afGe[0  , 0] := 1.00000E+01; afGe[0  , 1] := 8.81266E-03;
afGe[1  , 0] := 1.99800E+01; afGe[1  , 1] := 9.77619E-03;
afGe[2  , 0] := 2.99600E+01; afGe[2  , 1] := 9.38887E-01;
afGe[3  , 0] := 3.99400E+01; afGe[3  , 1] := 1.88885E+00;
afGe[4  , 0] := 4.99200E+01; afGe[4  , 1] := 3.37924E+00;
afGe[5  , 0] := 5.99000E+01; afGe[5  , 1] := 5.17287E+00;
afGe[6  , 0] := 6.98800E+01; afGe[6  , 1] := 6.99851E+00;
afGe[7  , 0] := 7.98600E+01; afGe[7  , 1] := 8.65575E+00;
afGe[8  , 0] := 8.98400E+01; afGe[8  , 1] := 1.00383E+01;
afGe[9  , 0] := 9.98200E+01; afGe[9  , 1] := 1.11123E+01;
afGe[10 , 0] := 1.09800E+02; afGe[10 , 1] := 1.18992E+01;
afGe[11 , 0] := 1.19780E+02; afGe[11 , 1] := 1.25300E+01;
afGe[12 , 0] := 1.29760E+02; afGe[12 , 1] := 1.31929E+01;
afGe[13 , 0] := 1.39740E+02; afGe[13 , 1] := 1.34683E+01;
afGe[14 , 0] := 1.49720E+02; afGe[14 , 1] := 1.35531E+01;
afGe[15 , 0] := 1.59700E+02; afGe[15 , 1] := 1.35254E+01;
afGe[16 , 0] := 1.69680E+02; afGe[16 , 1] := 1.34259E+01;
afGe[17 , 0] := 1.79660E+02; afGe[17 , 1] := 1.34620E+01;
afGe[18 , 0] := 1.89640E+02; afGe[18 , 1] := 1.35247E+01;
afGe[19 , 0] := 1.99620E+02; afGe[19 , 1] := 1.33231E+01;
afGe[20 , 0] := 2.09600E+02; afGe[20 , 1] := 1.30862E+01;
afGe[21 , 0] := 2.19580E+02; afGe[21 , 1] := 1.28308E+01;
afGe[22 , 0] := 2.29560E+02; afGe[22 , 1] := 1.25655E+01;
afGe[23 , 0] := 2.39540E+02; afGe[23 , 1] := 1.22951E+01;
afGe[24 , 0] := 2.49520E+02; afGe[24 , 1] := 1.20227E+01;
afGe[25 , 0] := 2.59500E+02; afGe[25 , 1] := 1.17524E+01;
afGe[26 , 0] := 2.69480E+02; afGe[26 , 1] := 1.14845E+01;
afGe[27 , 0] := 2.79460E+02; afGe[27 , 1] := 1.12208E+01;
afGe[28 , 0] := 2.89440E+02; afGe[28 , 1] := 1.09627E+01;
afGe[29 , 0] := 2.99420E+02; afGe[29 , 1] := 1.07107E+01;
afGe[30 , 0] := 3.09400E+02; afGe[30 , 1] := 1.04654E+01;
afGe[31 , 0] := 3.19380E+02; afGe[31 , 1] := 1.02271E+01;
afGe[32 , 0] := 3.29360E+02; afGe[32 , 1] := 9.99516E+00;
afGe[33 , 0] := 3.39340E+02; afGe[33 , 1] := 9.77038E+00;
afGe[34 , 0] := 3.49320E+02; afGe[34 , 1] := 9.55249E+00;
afGe[35 , 0] := 3.59300E+02; afGe[35 , 1] := 9.34153E+00;
afGe[36 , 0] := 3.69280E+02; afGe[36 , 1] := 9.13877E+00;
afGe[37 , 0] := 3.79260E+02; afGe[37 , 1] := 8.94103E+00;
afGe[38 , 0] := 3.89240E+02; afGe[38 , 1] := 8.75052E+00;
afGe[39 , 0] := 3.99220E+02; afGe[39 , 1] := 8.56542E+00;
afGe[40 , 0] := 4.09200E+02; afGe[40 , 1] := 8.38625E+00;
afGe[41 , 0] := 4.19180E+02; afGe[41 , 1] := 8.21293E+00;
afGe[42 , 0] := 4.29160E+02; afGe[42 , 1] := 8.04518E+00;
afGe[43 , 0] := 4.39140E+02; afGe[43 , 1] := 7.88279E+00;
afGe[44 , 0] := 4.49120E+02; afGe[44 , 1] := 7.72562E+00;
afGe[45 , 0] := 4.59100E+02; afGe[45 , 1] := 7.57349E+00;
afGe[46 , 0] := 4.69080E+02; afGe[46 , 1] := 7.42603E+00;
afGe[47 , 0] := 4.79060E+02; afGe[47 , 1] := 7.28323E+00;
afGe[48 , 0] := 4.89040E+02; afGe[48 , 1] := 7.14478E+00;
afGe[49 , 0] := 4.99020E+02; afGe[49 , 1] := 7.01042E+00;
afGe[50 , 0] := 5.09000E+02; afGe[50 , 1] := 6.87999E+00;
afGe[51 , 0] := 5.18980E+02; afGe[51 , 1] := 6.75328E+00;
afGe[52 , 0] := 5.28960E+02; afGe[52 , 1] := 6.63015E+00;
afGe[53 , 0] := 5.38940E+02; afGe[53 , 1] := 6.50950E+00;
afGe[54 , 0] := 5.48920E+02; afGe[54 , 1] := 6.37387E+00;
afGe[55 , 0] := 5.58900E+02; afGe[55 , 1] := 6.24150E+00;
afGe[56 , 0] := 5.68880E+02; afGe[56 , 1] := 6.11335E+00;
afGe[57 , 0] := 5.78860E+02; afGe[57 , 1] := 5.98927E+00;
afGe[58 , 0] := 5.88840E+02; afGe[58 , 1] := 5.86901E+00;
afGe[59 , 0] := 5.98820E+02; afGe[59 , 1] := 5.75252E+00;
afGe[60 , 0] := 6.08800E+02; afGe[60 , 1] := 5.63965E+00;
afGe[61 , 0] := 6.18780E+02; afGe[61 , 1] := 5.53035E+00;
afGe[62 , 0] := 6.28760E+02; afGe[62 , 1] := 5.42432E+00;
afGe[63 , 0] := 6.38740E+02; afGe[63 , 1] := 5.32161E+00;
afGe[64 , 0] := 6.48720E+02; afGe[64 , 1] := 5.22199E+00;
afGe[65 , 0] := 6.58700E+02; afGe[65 , 1] := 5.12538E+00;
afGe[66 , 0] := 6.68680E+02; afGe[66 , 1] := 5.03171E+00;
afGe[67 , 0] := 6.78660E+02; afGe[67 , 1] := 4.94078E+00;
afGe[68 , 0] := 6.88640E+02; afGe[68 , 1] := 4.85261E+00;
afGe[69 , 0] := 6.98620E+02; afGe[69 , 1] := 4.76709E+00;
afGe[70 , 0] := 7.08600E+02; afGe[70 , 1] := 4.68403E+00;
afGe[71 , 0] := 7.18580E+02; afGe[71 , 1] := 4.60334E+00;
afGe[72 , 0] := 7.28560E+02; afGe[72 , 1] := 4.52505E+00;
afGe[73 , 0] := 7.38540E+02; afGe[73 , 1] := 4.44896E+00;
afGe[74 , 0] := 7.48520E+02; afGe[74 , 1] := 4.37500E+00;
afGe[75 , 0] := 7.58500E+02; afGe[75 , 1] := 4.30316E+00;
afGe[76 , 0] := 7.68480E+02; afGe[76 , 1] := 4.23330E+00;
afGe[77 , 0] := 7.78460E+02; afGe[77 , 1] := 4.16541E+00;
afGe[78 , 0] := 7.88440E+02; afGe[78 , 1] := 4.09937E+00;
afGe[79 , 0] := 7.98420E+02; afGe[79 , 1] := 4.03513E+00;
afGe[80 , 0] := 8.08400E+02; afGe[80 , 1] := 3.97263E+00;
afGe[81 , 0] := 8.18380E+02; afGe[81 , 1] := 3.91191E+00;
afGe[82 , 0] := 8.28360E+02; afGe[82 , 1] := 3.85273E+00;
afGe[83 , 0] := 8.38340E+02; afGe[83 , 1] := 3.79513E+00;
afGe[84 , 0] := 8.48320E+02; afGe[84 , 1] := 3.73906E+00;
afGe[85 , 0] := 8.58300E+02; afGe[85 , 1] := 3.68448E+00;
afGe[86 , 0] := 8.68280E+02; afGe[86 , 1] := 3.63135E+00;
afGe[87 , 0] := 8.78260E+02; afGe[87 , 1] := 3.57961E+00;
afGe[88 , 0] := 8.88240E+02; afGe[88 , 1] := 3.52916E+00;
afGe[89 , 0] := 8.98220E+02; afGe[89 , 1] := 3.48008E+00;
afGe[90 , 0] := 9.08200E+02; afGe[90 , 1] := 3.43216E+00;
afGe[91 , 0] := 9.18180E+02; afGe[91 , 1] := 3.38550E+00;
afGe[92 , 0] := 9.28160E+02; afGe[92 , 1] := 3.34002E+00;
afGe[93 , 0] := 9.38140E+02; afGe[93 , 1] := 3.29570E+00;
afGe[94 , 0] := 9.48120E+02; afGe[94 , 1] := 3.25244E+00;
afGe[95 , 0] := 9.58100E+02; afGe[95 , 1] := 3.21028E+00;
afGe[96 , 0] := 9.68080E+02; afGe[96 , 1] := 3.16911E+00;
afGe[97 , 0] := 9.78060E+02; afGe[97 , 1] := 3.12900E+00;
afGe[98 , 0] := 9.88040E+02; afGe[98 , 1] := 3.08993E+00;
afGe[99 , 0] := 9.98020E+02; afGe[99 , 1] := 3.05154E+00;
afGe[100, 0] := 1.00800E+03; afGe[100, 1] := 3.00590E+00;
afGe[101, 0] := 1.01798E+03; afGe[101, 1] := 2.95919E+00;
afGe[102, 0] := 1.02796E+03; afGe[102, 1] := 2.91380E+00;
afGe[103, 0] := 1.03794E+03; afGe[103, 1] := 2.86980E+00;
afGe[104, 0] := 1.04792E+03; afGe[104, 1] := 2.82706E+00;
afGe[105, 0] := 1.05790E+03; afGe[105, 1] := 2.78554E+00;
afGe[106, 0] := 1.06788E+03; afGe[106, 1] := 2.74530E+00;
afGe[107, 0] := 1.07786E+03; afGe[107, 1] := 2.70625E+00;
afGe[108, 0] := 1.08784E+03; afGe[108, 1] := 2.66832E+00;
afGe[109, 0] := 1.09782E+03; afGe[109, 1] := 2.63157E+00;
afGe[110, 0] := 1.10780E+03; afGe[110, 1] := 2.59602E+00;
afGe[111, 0] := 1.11778E+03; afGe[111, 1] := 2.56169E+00;
afGe[112, 0] := 1.12776E+03; afGe[112, 1] := 2.52857E+00;
afGe[113, 0] := 1.13774E+03; afGe[113, 1] := 2.49676E+00;
afGe[114, 0] := 1.14772E+03; afGe[114, 1] := 2.46646E+00;
afGe[115, 0] := 1.15770E+03; afGe[115, 1] := 2.43792E+00;
afGe[116, 0] := 1.16768E+03; afGe[116, 1] := 2.41186E+00;
afGe[117, 0] := 1.17766E+03; afGe[117, 1] := 2.38937E+00;
afGe[118, 0] := 1.18764E+03; afGe[118, 1] := 2.37354E+00;
afGe[119, 0] := 1.19762E+03; afGe[119, 1] := 2.37603E+00;
afGe[120, 0] := 1.20760E+03; afGe[120, 1] := 2.42572E+00;
afGe[121, 0] := 1.21758E+03; afGe[121, 1] := 1.04902E+01;
afGe[122, 0] := 1.22756E+03; afGe[122, 1] := 1.16543E+01;
afGe[123, 0] := 1.23754E+03; afGe[123, 1] := 1.16089E+01;
afGe[124, 0] := 1.24752E+03; afGe[124, 1] := 1.32333E+01;
afGe[125, 0] := 1.25750E+03; afGe[125, 1] := 1.59139E+01;
afGe[126, 0] := 1.26748E+03; afGe[126, 1] := 1.57653E+01;
afGe[127, 0] := 1.27746E+03; afGe[127, 1] := 1.55814E+01;
afGe[128, 0] := 1.28744E+03; afGe[128, 1] := 1.53966E+01;
afGe[129, 0] := 1.29742E+03; afGe[129, 1] := 1.52130E+01;
afGe[130, 0] := 1.30740E+03; afGe[130, 1] := 1.50320E+01;
afGe[131, 0] := 1.31738E+03; afGe[131, 1] := 1.48540E+01;
afGe[132, 0] := 1.32736E+03; afGe[132, 1] := 1.46798E+01;
afGe[133, 0] := 1.33734E+03; afGe[133, 1] := 1.45095E+01;
afGe[134, 0] := 1.34732E+03; afGe[134, 1] := 1.43434E+01;
afGe[135, 0] := 1.35730E+03; afGe[135, 1] := 1.41819E+01;
afGe[136, 0] := 1.36728E+03; afGe[136, 1] := 1.40278E+01;
afGe[137, 0] := 1.37726E+03; afGe[137, 1] := 1.38825E+01;
afGe[138, 0] := 1.38724E+03; afGe[138, 1] := 1.37511E+01;
afGe[139, 0] := 1.39722E+03; afGe[139, 1] := 1.36552E+01;
afGe[140, 0] := 1.40720E+03; afGe[140, 1] := 1.38527E+01;
afGe[141, 0] := 1.41718E+03; afGe[141, 1] := 1.43567E+01;
afGe[142, 0] := 1.42716E+03; afGe[142, 1] := 1.46784E+01;
afGe[143, 0] := 1.43714E+03; afGe[143, 1] := 1.46147E+01;
afGe[144, 0] := 1.44712E+03; afGe[144, 1] := 1.45112E+01;
afGe[145, 0] := 1.45710E+03; afGe[145, 1] := 1.43870E+01;
afGe[146, 0] := 1.46708E+03; afGe[146, 1] := 1.42551E+01;
afGe[147, 0] := 1.47706E+03; afGe[147, 1] := 1.41225E+01;
afGe[148, 0] := 1.48704E+03; afGe[148, 1] := 1.39900E+01;
afGe[149, 0] := 1.49702E+03; afGe[149, 1] := 1.38582E+01;
afGe[150, 0] := 1.50700E+03; afGe[150, 1] := 1.37276E+01;
afGe[151, 0] := 1.51698E+03; afGe[151, 1] := 1.35987E+01;
afGe[152, 0] := 1.52696E+03; afGe[152, 1] := 1.34714E+01;
afGe[153, 0] := 1.53694E+03; afGe[153, 1] := 1.33454E+01;
afGe[154, 0] := 1.54692E+03; afGe[154, 1] := 1.32210E+01;
afGe[155, 0] := 1.55690E+03; afGe[155, 1] := 1.30993E+01;
afGe[156, 0] := 1.56688E+03; afGe[156, 1] := 1.29789E+01;
afGe[157, 0] := 1.57686E+03; afGe[157, 1] := 1.28599E+01;
afGe[158, 0] := 1.58684E+03; afGe[158, 1] := 1.27429E+01;
afGe[159, 0] := 1.59682E+03; afGe[159, 1] := 1.26273E+01;
afGe[160, 0] := 1.60680E+03; afGe[160, 1] := 1.25128E+01;
afGe[161, 0] := 1.61678E+03; afGe[161, 1] := 1.23997E+01;
afGe[162, 0] := 1.62676E+03; afGe[162, 1] := 1.22884E+01;
afGe[163, 0] := 1.63674E+03; afGe[163, 1] := 1.21789E+01;
afGe[164, 0] := 1.64672E+03; afGe[164, 1] := 1.20708E+01;
afGe[165, 0] := 1.65670E+03; afGe[165, 1] := 1.19641E+01;
afGe[166, 0] := 1.66668E+03; afGe[166, 1] := 1.18588E+01;
afGe[167, 0] := 1.67666E+03; afGe[167, 1] := 1.17550E+01;
afGe[168, 0] := 1.68664E+03; afGe[168, 1] := 1.16530E+01;
afGe[169, 0] := 1.69662E+03; afGe[169, 1] := 1.15522E+01;
afGe[170, 0] := 1.70660E+03; afGe[170, 1] := 1.14528E+01;
afGe[171, 0] := 1.71658E+03; afGe[171, 1] := 1.13551E+01;
afGe[172, 0] := 1.72656E+03; afGe[172, 1] := 1.12588E+01;
afGe[173, 0] := 1.73654E+03; afGe[173, 1] := 1.11637E+01;
afGe[174, 0] := 1.74652E+03; afGe[174, 1] := 1.10701E+01;
afGe[175, 0] := 1.75650E+03; afGe[175, 1] := 1.09779E+01;
afGe[176, 0] := 1.76648E+03; afGe[176, 1] := 1.08865E+01;
afGe[177, 0] := 1.77646E+03; afGe[177, 1] := 1.07962E+01;
afGe[178, 0] := 1.78644E+03; afGe[178, 1] := 1.07080E+01;
afGe[179, 0] := 1.79642E+03; afGe[179, 1] := 1.06210E+01;
afGe[180, 0] := 1.80640E+03; afGe[180, 1] := 1.05345E+01;
afGe[181, 0] := 1.81638E+03; afGe[181, 1] := 1.04494E+01;
afGe[182, 0] := 1.82636E+03; afGe[182, 1] := 1.03656E+01;
afGe[183, 0] := 1.83634E+03; afGe[183, 1] := 1.02827E+01;
afGe[184, 0] := 1.84632E+03; afGe[184, 1] := 1.02005E+01;
afGe[185, 0] := 1.85630E+03; afGe[185, 1] := 1.01190E+01;
afGe[186, 0] := 1.86628E+03; afGe[186, 1] := 1.00383E+01;
afGe[187, 0] := 1.87626E+03; afGe[187, 1] := 9.95872E+00;
afGe[188, 0] := 1.88624E+03; afGe[188, 1] := 9.88014E+00;
afGe[189, 0] := 1.89622E+03; afGe[189, 1] := 9.80266E+00;
afGe[190, 0] := 1.90620E+03; afGe[190, 1] := 9.72617E+00;
afGe[191, 0] := 1.91618E+03; afGe[191, 1] := 9.65061E+00;
afGe[192, 0] := 1.92616E+03; afGe[192, 1] := 9.57603E+00;
afGe[193, 0] := 1.93614E+03; afGe[193, 1] := 9.50244E+00;
afGe[194, 0] := 1.94612E+03; afGe[194, 1] := 9.42979E+00;
afGe[195, 0] := 1.95610E+03; afGe[195, 1] := 9.35802E+00;
afGe[196, 0] := 1.96608E+03; afGe[196, 1] := 9.28715E+00;
afGe[197, 0] := 1.97606E+03; afGe[197, 1] := 9.21715E+00;
afGe[198, 0] := 1.98604E+03; afGe[198, 1] := 9.14804E+00;
afGe[199, 0] := 1.99602E+03; afGe[199, 1] := 9.07981E+00;
afGe[200, 0] := 2.00600E+03; afGe[200, 1] := 9.01242E+00;
afGe[201, 0] := 2.01598E+03; afGe[201, 1] := 8.94582E+00;
afGe[202, 0] := 2.02596E+03; afGe[202, 1] := 8.88005E+00;
afGe[203, 0] := 2.03594E+03; afGe[203, 1] := 8.81508E+00;
afGe[204, 0] := 2.04592E+03; afGe[204, 1] := 8.75091E+00;
afGe[205, 0] := 2.05590E+03; afGe[205, 1] := 8.68749E+00;
afGe[206, 0] := 2.06588E+03; afGe[206, 1] := 8.62505E+00;
afGe[207, 0] := 2.07586E+03; afGe[207, 1] := 8.56388E+00;
afGe[208, 0] := 2.08584E+03; afGe[208, 1] := 8.50327E+00;
afGe[209, 0] := 2.09582E+03; afGe[209, 1] := 8.44283E+00;
afGe[210, 0] := 2.10580E+03; afGe[210, 1] := 8.38315E+00;
afGe[211, 0] := 2.11578E+03; afGe[211, 1] := 8.32444E+00;
afGe[212, 0] := 2.12576E+03; afGe[212, 1] := 8.26640E+00;
afGe[213, 0] := 2.13574E+03; afGe[213, 1] := 8.20872E+00;
afGe[214, 0] := 2.14572E+03; afGe[214, 1] := 8.15170E+00;
afGe[215, 0] := 2.15570E+03; afGe[215, 1] := 8.09537E+00;
afGe[216, 0] := 2.16568E+03; afGe[216, 1] := 8.03970E+00;
afGe[217, 0] := 2.17566E+03; afGe[217, 1] := 7.98464E+00;
afGe[218, 0] := 2.18564E+03; afGe[218, 1] := 7.93020E+00;
afGe[219, 0] := 2.19562E+03; afGe[219, 1] := 7.87639E+00;
afGe[220, 0] := 2.20560E+03; afGe[220, 1] := 7.82319E+00;
afGe[221, 0] := 2.21558E+03; afGe[221, 1] := 7.77059E+00;
afGe[222, 0] := 2.22556E+03; afGe[222, 1] := 7.71857E+00;
afGe[223, 0] := 2.23554E+03; afGe[223, 1] := 7.66714E+00;
afGe[224, 0] := 2.24552E+03; afGe[224, 1] := 7.61631E+00;
afGe[225, 0] := 2.25550E+03; afGe[225, 1] := 7.56604E+00;
afGe[226, 0] := 2.26548E+03; afGe[226, 1] := 7.51609E+00;
afGe[227, 0] := 2.27546E+03; afGe[227, 1] := 7.46667E+00;
afGe[228, 0] := 2.28544E+03; afGe[228, 1] := 7.41759E+00;
afGe[229, 0] := 2.29542E+03; afGe[229, 1] := 7.36895E+00;
afGe[230, 0] := 2.30540E+03; afGe[230, 1] := 7.32086E+00;
afGe[231, 0] := 2.31538E+03; afGe[231, 1] := 7.27333E+00;
afGe[232, 0] := 2.32536E+03; afGe[232, 1] := 7.22631E+00;
afGe[233, 0] := 2.33534E+03; afGe[233, 1] := 7.17978E+00;
afGe[234, 0] := 2.34532E+03; afGe[234, 1] := 7.13374E+00;
afGe[235, 0] := 2.35530E+03; afGe[235, 1] := 7.08820E+00;
afGe[236, 0] := 2.36528E+03; afGe[236, 1] := 7.04313E+00;
afGe[237, 0] := 2.37526E+03; afGe[237, 1] := 6.99855E+00;
afGe[238, 0] := 2.38524E+03; afGe[238, 1] := 6.95443E+00;
afGe[239, 0] := 2.39522E+03; afGe[239, 1] := 6.91078E+00;
afGe[240, 0] := 2.40520E+03; afGe[240, 1] := 6.86747E+00;
afGe[241, 0] := 2.41518E+03; afGe[241, 1] := 6.82461E+00;
afGe[242, 0] := 2.42516E+03; afGe[242, 1] := 6.78179E+00;
afGe[243, 0] := 2.43514E+03; afGe[243, 1] := 6.73917E+00;
afGe[244, 0] := 2.44512E+03; afGe[244, 1] := 6.69685E+00;
afGe[245, 0] := 2.45510E+03; afGe[245, 1] := 6.65438E+00;
afGe[246, 0] := 2.46508E+03; afGe[246, 1] := 6.61235E+00;
afGe[247, 0] := 2.47506E+03; afGe[247, 1] := 6.57073E+00;
afGe[248, 0] := 2.48504E+03; afGe[248, 1] := 6.52952E+00;
afGe[249, 0] := 2.49502E+03; afGe[249, 1] := 6.48860E+00;
afGe[250, 0] := 2.50500E+03; afGe[250, 1] := 6.44771E+00;
afGe[251, 0] := 2.51498E+03; afGe[251, 1] := 6.40725E+00;
afGe[252, 0] := 2.52496E+03; afGe[252, 1] := 6.36714E+00;
afGe[253, 0] := 2.53494E+03; afGe[253, 1] := 6.32742E+00;
afGe[254, 0] := 2.54492E+03; afGe[254, 1] := 6.28811E+00;
afGe[255, 0] := 2.55490E+03; afGe[255, 1] := 6.24920E+00;
afGe[256, 0] := 2.56488E+03; afGe[256, 1] := 6.21069E+00;
afGe[257, 0] := 2.57486E+03; afGe[257, 1] := 6.17257E+00;
afGe[258, 0] := 2.58484E+03; afGe[258, 1] := 6.13484E+00;
afGe[259, 0] := 2.59482E+03; afGe[259, 1] := 6.09749E+00;
afGe[260, 0] := 2.60480E+03; afGe[260, 1] := 6.06050E+00;
afGe[261, 0] := 2.61478E+03; afGe[261, 1] := 6.02387E+00;
afGe[262, 0] := 2.62476E+03; afGe[262, 1] := 5.98760E+00;
afGe[263, 0] := 2.63474E+03; afGe[263, 1] := 5.95169E+00;
afGe[264, 0] := 2.64472E+03; afGe[264, 1] := 5.91613E+00;
afGe[265, 0] := 2.65470E+03; afGe[265, 1] := 5.88096E+00;
afGe[266, 0] := 2.66468E+03; afGe[266, 1] := 5.84614E+00;
afGe[267, 0] := 2.67466E+03; afGe[267, 1] := 5.81165E+00;
afGe[268, 0] := 2.68464E+03; afGe[268, 1] := 5.77751E+00;
afGe[269, 0] := 2.69462E+03; afGe[269, 1] := 5.74370E+00;
afGe[270, 0] := 2.70460E+03; afGe[270, 1] := 5.71023E+00;
afGe[271, 0] := 2.71458E+03; afGe[271, 1] := 5.67708E+00;
afGe[272, 0] := 2.72456E+03; afGe[272, 1] := 5.64425E+00;
afGe[273, 0] := 2.73454E+03; afGe[273, 1] := 5.61173E+00;
afGe[274, 0] := 2.74452E+03; afGe[274, 1] := 5.57952E+00;
afGe[275, 0] := 2.75450E+03; afGe[275, 1] := 5.54761E+00;
afGe[276, 0] := 2.76448E+03; afGe[276, 1] := 5.51604E+00;
afGe[277, 0] := 2.77446E+03; afGe[277, 1] := 5.48476E+00;
afGe[278, 0] := 2.78444E+03; afGe[278, 1] := 5.45377E+00;
afGe[279, 0] := 2.79442E+03; afGe[279, 1] := 5.42305E+00;
afGe[280, 0] := 2.80440E+03; afGe[280, 1] := 5.39261E+00;
afGe[281, 0] := 2.81438E+03; afGe[281, 1] := 5.36242E+00;
afGe[282, 0] := 2.82436E+03; afGe[282, 1] := 5.33248E+00;
afGe[283, 0] := 2.83434E+03; afGe[283, 1] := 5.30282E+00;
afGe[284, 0] := 2.84432E+03; afGe[284, 1] := 5.27320E+00;
afGe[285, 0] := 2.85430E+03; afGe[285, 1] := 5.24379E+00;
afGe[286, 0] := 2.86428E+03; afGe[286, 1] := 5.21464E+00;
afGe[287, 0] := 2.87426E+03; afGe[287, 1] := 5.18575E+00;
afGe[288, 0] := 2.88424E+03; afGe[288, 1] := 5.15712E+00;
afGe[289, 0] := 2.89422E+03; afGe[289, 1] := 5.12874E+00;
afGe[290, 0] := 2.90420E+03; afGe[290, 1] := 5.10066E+00;
afGe[291, 0] := 2.91418E+03; afGe[291, 1] := 5.07282E+00;
afGe[292, 0] := 2.92416E+03; afGe[292, 1] := 5.04524E+00;
afGe[293, 0] := 2.93414E+03; afGe[293, 1] := 5.01794E+00;
afGe[294, 0] := 2.94412E+03; afGe[294, 1] := 4.99087E+00;
afGe[295, 0] := 2.95410E+03; afGe[295, 1] := 4.96405E+00;
afGe[296, 0] := 2.96408E+03; afGe[296, 1] := 4.93747E+00;
afGe[297, 0] := 2.97406E+03; afGe[297, 1] := 4.91113E+00;
afGe[298, 0] := 2.98404E+03; afGe[298, 1] := 4.88472E+00;
afGe[299, 0] := 2.99402E+03; afGe[299, 1] := 4.85784E+00;
afGe[300, 0] := 3.00400E+03; afGe[300, 1] := 4.83120E+00;
afGe[301, 0] := 3.01398E+03; afGe[301, 1] := 4.80425E+00;
afGe[302, 0] := 3.02396E+03; afGe[302, 1] := 4.77633E+00;
afGe[303, 0] := 3.03394E+03; afGe[303, 1] := 4.74867E+00;
afGe[304, 0] := 3.04392E+03; afGe[304, 1] := 4.72127E+00;
afGe[305, 0] := 3.05390E+03; afGe[305, 1] := 4.69418E+00;
afGe[306, 0] := 3.06388E+03; afGe[306, 1] := 4.66734E+00;
afGe[307, 0] := 3.07386E+03; afGe[307, 1] := 4.64073E+00;
afGe[308, 0] := 3.08384E+03; afGe[308, 1] := 4.61436E+00;
afGe[309, 0] := 3.09382E+03; afGe[309, 1] := 4.58821E+00;
afGe[310, 0] := 3.10380E+03; afGe[310, 1] := 4.56231E+00;
afGe[311, 0] := 3.11378E+03; afGe[311, 1] := 4.53666E+00;
afGe[312, 0] := 3.12376E+03; afGe[312, 1] := 4.51124E+00;
afGe[313, 0] := 3.13374E+03; afGe[313, 1] := 4.48604E+00;
afGe[314, 0] := 3.14372E+03; afGe[314, 1] := 4.46111E+00;
afGe[315, 0] := 3.15370E+03; afGe[315, 1] := 4.43639E+00;
afGe[316, 0] := 3.16368E+03; afGe[316, 1] := 4.41188E+00;
afGe[317, 0] := 3.17366E+03; afGe[317, 1] := 4.38761E+00;
afGe[318, 0] := 3.18364E+03; afGe[318, 1] := 4.36354E+00;
afGe[319, 0] := 3.19362E+03; afGe[319, 1] := 4.33968E+00;
afGe[320, 0] := 3.20360E+03; afGe[320, 1] := 4.31605E+00;
afGe[321, 0] := 3.21358E+03; afGe[321, 1] := 4.29262E+00;
afGe[322, 0] := 3.22356E+03; afGe[322, 1] := 4.26939E+00;
afGe[323, 0] := 3.23354E+03; afGe[323, 1] := 4.24638E+00;
afGe[324, 0] := 3.24352E+03; afGe[324, 1] := 4.22358E+00;
afGe[325, 0] := 3.25350E+03; afGe[325, 1] := 4.20097E+00;
afGe[326, 0] := 3.26348E+03; afGe[326, 1] := 4.17855E+00;
afGe[327, 0] := 3.27346E+03; afGe[327, 1] := 4.15633E+00;
afGe[328, 0] := 3.28344E+03; afGe[328, 1] := 4.13429E+00;
afGe[329, 0] := 3.29342E+03; afGe[329, 1] := 4.11244E+00;
afGe[330, 0] := 3.30340E+03; afGe[330, 1] := 4.09082E+00;
afGe[331, 0] := 3.31338E+03; afGe[331, 1] := 4.06937E+00;
afGe[332, 0] := 3.32336E+03; afGe[332, 1] := 4.04810E+00;
afGe[333, 0] := 3.33334E+03; afGe[333, 1] := 4.02700E+00;
afGe[334, 0] := 3.34332E+03; afGe[334, 1] := 4.00608E+00;
afGe[335, 0] := 3.35330E+03; afGe[335, 1] := 3.98532E+00;
afGe[336, 0] := 3.36328E+03; afGe[336, 1] := 3.96475E+00;
afGe[337, 0] := 3.37326E+03; afGe[337, 1] := 3.94436E+00;
afGe[338, 0] := 3.38324E+03; afGe[338, 1] := 3.92413E+00;
afGe[339, 0] := 3.39322E+03; afGe[339, 1] := 3.90407E+00;
afGe[340, 0] := 3.40320E+03; afGe[340, 1] := 3.88412E+00;
afGe[341, 0] := 3.41318E+03; afGe[341, 1] := 3.86433E+00;
afGe[342, 0] := 3.42316E+03; afGe[342, 1] := 3.84469E+00;
afGe[343, 0] := 3.43314E+03; afGe[343, 1] := 3.82522E+00;
afGe[344, 0] := 3.44312E+03; afGe[344, 1] := 3.80592E+00;
afGe[345, 0] := 3.45310E+03; afGe[345, 1] := 3.78676E+00;
afGe[346, 0] := 3.46308E+03; afGe[346, 1] := 3.76776E+00;
afGe[347, 0] := 3.47306E+03; afGe[347, 1] := 3.74896E+00;
afGe[348, 0] := 3.48304E+03; afGe[348, 1] := 3.73030E+00;
afGe[349, 0] := 3.49302E+03; afGe[349, 1] := 3.71178E+00;
afGe[350, 0] := 3.50300E+03; afGe[350, 1] := 3.69341E+00;
afGe[351, 0] := 3.51298E+03; afGe[351, 1] := 3.67518E+00;
afGe[352, 0] := 3.52296E+03; afGe[352, 1] := 3.65709E+00;
afGe[353, 0] := 3.53294E+03; afGe[353, 1] := 3.63915E+00;
afGe[354, 0] := 3.54292E+03; afGe[354, 1] := 3.62137E+00;
afGe[355, 0] := 3.55290E+03; afGe[355, 1] := 3.60373E+00;
afGe[356, 0] := 3.56288E+03; afGe[356, 1] := 3.58622E+00;
afGe[357, 0] := 3.57286E+03; afGe[357, 1] := 3.56888E+00;
afGe[358, 0] := 3.58284E+03; afGe[358, 1] := 3.55167E+00;
afGe[359, 0] := 3.59282E+03; afGe[359, 1] := 3.53460E+00;
afGe[360, 0] := 3.60280E+03; afGe[360, 1] := 3.51765E+00;
afGe[361, 0] := 3.61278E+03; afGe[361, 1] := 3.50082E+00;
afGe[362, 0] := 3.62276E+03; afGe[362, 1] := 3.48412E+00;
afGe[363, 0] := 3.63274E+03; afGe[363, 1] := 3.46754E+00;
afGe[364, 0] := 3.64272E+03; afGe[364, 1] := 3.45111E+00;
afGe[365, 0] := 3.65270E+03; afGe[365, 1] := 3.43483E+00;
afGe[366, 0] := 3.66268E+03; afGe[366, 1] := 3.41866E+00;
afGe[367, 0] := 3.67266E+03; afGe[367, 1] := 3.40262E+00;
afGe[368, 0] := 3.68264E+03; afGe[368, 1] := 3.38669E+00;
afGe[369, 0] := 3.69262E+03; afGe[369, 1] := 3.37089E+00;
afGe[370, 0] := 3.70260E+03; afGe[370, 1] := 3.35519E+00;
afGe[371, 0] := 3.71258E+03; afGe[371, 1] := 3.33962E+00;
afGe[372, 0] := 3.72256E+03; afGe[372, 1] := 3.32419E+00;
afGe[373, 0] := 3.73254E+03; afGe[373, 1] := 3.30887E+00;
afGe[374, 0] := 3.74252E+03; afGe[374, 1] := 3.29365E+00;
afGe[375, 0] := 3.75250E+03; afGe[375, 1] := 3.27856E+00;
afGe[376, 0] := 3.76248E+03; afGe[376, 1] := 3.26358E+00;
afGe[377, 0] := 3.77246E+03; afGe[377, 1] := 3.24870E+00;
afGe[378, 0] := 3.78244E+03; afGe[378, 1] := 3.23393E+00;
afGe[379, 0] := 3.79242E+03; afGe[379, 1] := 3.21928E+00;
afGe[380, 0] := 3.80240E+03; afGe[380, 1] := 3.20474E+00;
afGe[381, 0] := 3.81238E+03; afGe[381, 1] := 3.19030E+00;
afGe[382, 0] := 3.82236E+03; afGe[382, 1] := 3.17596E+00;
afGe[383, 0] := 3.83234E+03; afGe[383, 1] := 3.16174E+00;
afGe[384, 0] := 3.84232E+03; afGe[384, 1] := 3.14762E+00;
afGe[385, 0] := 3.85230E+03; afGe[385, 1] := 3.13360E+00;
afGe[386, 0] := 3.86228E+03; afGe[386, 1] := 3.11968E+00;
afGe[387, 0] := 3.87226E+03; afGe[387, 1] := 3.10588E+00;
afGe[388, 0] := 3.88224E+03; afGe[388, 1] := 3.09218E+00;
afGe[389, 0] := 3.89222E+03; afGe[389, 1] := 3.07857E+00;
afGe[390, 0] := 3.90220E+03; afGe[390, 1] := 3.06506E+00;
afGe[391, 0] := 3.91218E+03; afGe[391, 1] := 3.05166E+00;
afGe[392, 0] := 3.92216E+03; afGe[392, 1] := 3.03836E+00;
afGe[393, 0] := 3.93214E+03; afGe[393, 1] := 3.02515E+00;
afGe[394, 0] := 3.94212E+03; afGe[394, 1] := 3.01203E+00;
afGe[395, 0] := 3.95210E+03; afGe[395, 1] := 2.99901E+00;
afGe[396, 0] := 3.96208E+03; afGe[396, 1] := 2.98608E+00;
afGe[397, 0] := 3.97206E+03; afGe[397, 1] := 2.97323E+00;
afGe[398, 0] := 3.98204E+03; afGe[398, 1] := 2.96047E+00;
afGe[399, 0] := 3.99202E+03; afGe[399, 1] := 2.94781E+00;
afGe[400, 0] := 4.00200E+03; afGe[400, 1] := 2.93523E+00;
afGe[401, 0] := 4.01198E+03; afGe[401, 1] := 2.92274E+00;
afGe[402, 0] := 4.02196E+03; afGe[402, 1] := 2.91033E+00;
afGe[403, 0] := 4.03194E+03; afGe[403, 1] := 2.89802E+00;
afGe[404, 0] := 4.04192E+03; afGe[404, 1] := 2.88579E+00;
afGe[405, 0] := 4.05190E+03; afGe[405, 1] := 2.87364E+00;
afGe[406, 0] := 4.06188E+03; afGe[406, 1] := 2.86158E+00;
afGe[407, 0] := 4.07186E+03; afGe[407, 1] := 2.84961E+00;
afGe[408, 0] := 4.08184E+03; afGe[408, 1] := 2.83772E+00;
afGe[409, 0] := 4.09182E+03; afGe[409, 1] := 2.82591E+00;
afGe[410, 0] := 4.10180E+03; afGe[410, 1] := 2.81418E+00;
afGe[411, 0] := 4.11178E+03; afGe[411, 1] := 2.80254E+00;
afGe[412, 0] := 4.12176E+03; afGe[412, 1] := 2.79098E+00;
afGe[413, 0] := 4.13174E+03; afGe[413, 1] := 2.77950E+00;
afGe[414, 0] := 4.14172E+03; afGe[414, 1] := 2.76809E+00;
afGe[415, 0] := 4.15170E+03; afGe[415, 1] := 2.75678E+00;
afGe[416, 0] := 4.16168E+03; afGe[416, 1] := 2.74554E+00;
afGe[417, 0] := 4.17166E+03; afGe[417, 1] := 2.73438E+00;
afGe[418, 0] := 4.18164E+03; afGe[418, 1] := 2.72329E+00;
afGe[419, 0] := 4.19162E+03; afGe[419, 1] := 2.71224E+00;
afGe[420, 0] := 4.20160E+03; afGe[420, 1] := 2.70127E+00;
afGe[421, 0] := 4.21158E+03; afGe[421, 1] := 2.69037E+00;
afGe[422, 0] := 4.22156E+03; afGe[422, 1] := 2.67954E+00;
afGe[423, 0] := 4.23154E+03; afGe[423, 1] := 2.66881E+00;
afGe[424, 0] := 4.24152E+03; afGe[424, 1] := 2.65814E+00;
afGe[425, 0] := 4.25150E+03; afGe[425, 1] := 2.64755E+00;
afGe[426, 0] := 4.26148E+03; afGe[426, 1] := 2.63702E+00;
afGe[427, 0] := 4.27146E+03; afGe[427, 1] := 2.62657E+00;
afGe[428, 0] := 4.28144E+03; afGe[428, 1] := 2.61618E+00;
afGe[429, 0] := 4.29142E+03; afGe[429, 1] := 2.60586E+00;
afGe[430, 0] := 4.30140E+03; afGe[430, 1] := 2.59561E+00;
afGe[431, 0] := 4.31138E+03; afGe[431, 1] := 2.58542E+00;
afGe[432, 0] := 4.32136E+03; afGe[432, 1] := 2.57531E+00;
afGe[433, 0] := 4.33134E+03; afGe[433, 1] := 2.56526E+00;
afGe[434, 0] := 4.34132E+03; afGe[434, 1] := 2.55527E+00;
afGe[435, 0] := 4.35130E+03; afGe[435, 1] := 2.54534E+00;
afGe[436, 0] := 4.36128E+03; afGe[436, 1] := 2.53550E+00;
afGe[437, 0] := 4.37126E+03; afGe[437, 1] := 2.52571E+00;
afGe[438, 0] := 4.38124E+03; afGe[438, 1] := 2.51598E+00;
afGe[439, 0] := 4.39122E+03; afGe[439, 1] := 2.50632E+00;
afGe[440, 0] := 4.40120E+03; afGe[440, 1] := 2.49670E+00;
afGe[441, 0] := 4.41118E+03; afGe[441, 1] := 2.48715E+00;
afGe[442, 0] := 4.42116E+03; afGe[442, 1] := 2.47766E+00;
afGe[443, 0] := 4.43114E+03; afGe[443, 1] := 2.46822E+00;
afGe[444, 0] := 4.44112E+03; afGe[444, 1] := 2.45885E+00;
afGe[445, 0] := 4.45110E+03; afGe[445, 1] := 2.44955E+00;
afGe[446, 0] := 4.46108E+03; afGe[446, 1] := 2.44030E+00;
afGe[447, 0] := 4.47106E+03; afGe[447, 1] := 2.43111E+00;
afGe[448, 0] := 4.48104E+03; afGe[448, 1] := 2.42198E+00;
afGe[449, 0] := 4.49102E+03; afGe[449, 1] := 2.41290E+00;
afGe[450, 0] := 4.50100E+03; afGe[450, 1] := 2.40388E+00;
afGe[451, 0] := 4.51098E+03; afGe[451, 1] := 2.39492E+00;
afGe[452, 0] := 4.52096E+03; afGe[452, 1] := 2.38600E+00;
afGe[453, 0] := 4.53094E+03; afGe[453, 1] := 2.37714E+00;
afGe[454, 0] := 4.54092E+03; afGe[454, 1] := 2.36834E+00;
afGe[455, 0] := 4.55090E+03; afGe[455, 1] := 2.35959E+00;
afGe[456, 0] := 4.56088E+03; afGe[456, 1] := 2.35089E+00;
afGe[457, 0] := 4.57086E+03; afGe[457, 1] := 2.34224E+00;
afGe[458, 0] := 4.58084E+03; afGe[458, 1] := 2.33366E+00;
afGe[459, 0] := 4.59082E+03; afGe[459, 1] := 2.32515E+00;
afGe[460, 0] := 4.60080E+03; afGe[460, 1] := 2.31668E+00;
afGe[461, 0] := 4.61078E+03; afGe[461, 1] := 2.30826E+00;
afGe[462, 0] := 4.62076E+03; afGe[462, 1] := 2.29989E+00;
afGe[463, 0] := 4.63074E+03; afGe[463, 1] := 2.29156E+00;
afGe[464, 0] := 4.64072E+03; afGe[464, 1] := 2.28328E+00;
afGe[465, 0] := 4.65070E+03; afGe[465, 1] := 2.27504E+00;
afGe[466, 0] := 4.66068E+03; afGe[466, 1] := 2.26685E+00;
afGe[467, 0] := 4.67066E+03; afGe[467, 1] := 2.25872E+00;
afGe[468, 0] := 4.68064E+03; afGe[468, 1] := 2.25064E+00;
afGe[469, 0] := 4.69062E+03; afGe[469, 1] := 2.24261E+00;
afGe[470, 0] := 4.70060E+03; afGe[470, 1] := 2.23462E+00;
afGe[471, 0] := 4.71058E+03; afGe[471, 1] := 2.22667E+00;
afGe[472, 0] := 4.72056E+03; afGe[472, 1] := 2.21879E+00;
afGe[473, 0] := 4.73054E+03; afGe[473, 1] := 2.21095E+00;
afGe[474, 0] := 4.74052E+03; afGe[474, 1] := 2.20316E+00;
afGe[475, 0] := 4.75050E+03; afGe[475, 1] := 2.19541E+00;
afGe[476, 0] := 4.76048E+03; afGe[476, 1] := 2.18771E+00;
afGe[477, 0] := 4.77046E+03; afGe[477, 1] := 2.18004E+00;
afGe[478, 0] := 4.78044E+03; afGe[478, 1] := 2.17242E+00;
afGe[479, 0] := 4.79042E+03; afGe[479, 1] := 2.16484E+00;
afGe[480, 0] := 4.80040E+03; afGe[480, 1] := 2.15730E+00;
afGe[481, 0] := 4.81038E+03; afGe[481, 1] := 2.14982E+00;
afGe[482, 0] := 4.82036E+03; afGe[482, 1] := 2.14239E+00;
afGe[483, 0] := 4.83034E+03; afGe[483, 1] := 2.13499E+00;
afGe[484, 0] := 4.84032E+03; afGe[484, 1] := 2.12764E+00;
afGe[485, 0] := 4.85030E+03; afGe[485, 1] := 2.12033E+00;
afGe[486, 0] := 4.86028E+03; afGe[486, 1] := 2.11308E+00;
afGe[487, 0] := 4.87026E+03; afGe[487, 1] := 2.10587E+00;
afGe[488, 0] := 4.88024E+03; afGe[488, 1] := 2.09870E+00;
afGe[489, 0] := 4.89022E+03; afGe[489, 1] := 2.09157E+00;
afGe[490, 0] := 4.90020E+03; afGe[490, 1] := 2.08449E+00;
afGe[491, 0] := 4.91018E+03; afGe[491, 1] := 2.07742E+00;
afGe[492, 0] := 4.92016E+03; afGe[492, 1] := 2.07039E+00;
afGe[493, 0] := 4.93014E+03; afGe[493, 1] := 2.06340E+00;
afGe[494, 0] := 4.94012E+03; afGe[494, 1] := 2.05645E+00;
afGe[495, 0] := 4.95010E+03; afGe[495, 1] := 2.04954E+00;
afGe[496, 0] := 4.96008E+03; afGe[496, 1] := 2.04267E+00;
afGe[497, 0] := 4.97006E+03; afGe[497, 1] := 2.03583E+00;
afGe[498, 0] := 4.98004E+03; afGe[498, 1] := 2.02903E+00;
afGe[499, 0] := 4.99002E+03; afGe[499, 1] := 2.02227E+00;
afGe[500, 0] := 5.00000E+03; afGe[500, 1] := 2.01555E+00;
afGe[501, 0] := 5.05000E+03; afGe[501, 1] := 1.98243E+00;
afGe[502, 0] := 5.10000E+03; afGe[502, 1] := 1.95023E+00;
afGe[503, 0] := 5.15000E+03; afGe[503, 1] := 1.91893E+00;
afGe[504, 0] := 5.20000E+03; afGe[504, 1] := 1.88849E+00;
afGe[505, 0] := 5.25000E+03; afGe[505, 1] := 1.85882E+00;
afGe[506, 0] := 5.30000E+03; afGe[506, 1] := 1.82914E+00;
afGe[507, 0] := 5.35000E+03; afGe[507, 1] := 1.79992E+00;
afGe[508, 0] := 5.40000E+03; afGe[508, 1] := 1.77131E+00;
afGe[509, 0] := 5.45000E+03; afGe[509, 1] := 1.74311E+00;
afGe[510, 0] := 5.50000E+03; afGe[510, 1] := 1.71554E+00;
afGe[511, 0] := 5.55000E+03; afGe[511, 1] := 1.68867E+00;
afGe[512, 0] := 5.60000E+03; afGe[512, 1] := 1.66244E+00;
afGe[513, 0] := 5.65000E+03; afGe[513, 1] := 1.63688E+00;
afGe[514, 0] := 5.70000E+03; afGe[514, 1] := 1.61200E+00;
afGe[515, 0] := 5.75000E+03; afGe[515, 1] := 1.58772E+00;
afGe[516, 0] := 5.80000E+03; afGe[516, 1] := 1.56412E+00;
afGe[517, 0] := 5.85000E+03; afGe[517, 1] := 1.54110E+00;
afGe[518, 0] := 5.90000E+03; afGe[518, 1] := 1.51858E+00;
afGe[519, 0] := 5.95000E+03; afGe[519, 1] := 1.49663E+00;
afGe[520, 0] := 6.00000E+03; afGe[520, 1] := 1.47522E+00;
afGe[521, 0] := 6.05000E+03; afGe[521, 1] := 1.45429E+00;
afGe[522, 0] := 6.10000E+03; afGe[522, 1] := 1.43388E+00;
afGe[523, 0] := 6.15000E+03; afGe[523, 1] := 1.41343E+00;
afGe[524, 0] := 6.20000E+03; afGe[524, 1] := 1.39315E+00;
afGe[525, 0] := 6.25000E+03; afGe[525, 1] := 1.37325E+00;
afGe[526, 0] := 6.30000E+03; afGe[526, 1] := 1.35381E+00;
afGe[527, 0] := 6.35000E+03; afGe[527, 1] := 1.33477E+00;
afGe[528, 0] := 6.40000E+03; afGe[528, 1] := 1.31621E+00;
afGe[529, 0] := 6.45000E+03; afGe[529, 1] := 1.29804E+00;
afGe[530, 0] := 6.50000E+03; afGe[530, 1] := 1.28029E+00;
afGe[531, 0] := 6.55000E+03; afGe[531, 1] := 1.26295E+00;
afGe[532, 0] := 6.60000E+03; afGe[532, 1] := 1.24590E+00;
afGe[533, 0] := 6.65000E+03; afGe[533, 1] := 1.22928E+00;
afGe[534, 0] := 6.70000E+03; afGe[534, 1] := 1.21302E+00;
afGe[535, 0] := 6.75000E+03; afGe[535, 1] := 1.19711E+00;
afGe[536, 0] := 6.80000E+03; afGe[536, 1] := 1.18153E+00;
afGe[537, 0] := 6.85000E+03; afGe[537, 1] := 1.16629E+00;
afGe[538, 0] := 6.90000E+03; afGe[538, 1] := 1.15138E+00;
afGe[539, 0] := 6.95000E+03; afGe[539, 1] := 1.13677E+00;
afGe[540, 0] := 7.00000E+03; afGe[540, 1] := 1.12249E+00;
afGe[541, 0] := 7.05000E+03; afGe[541, 1] := 1.10846E+00;
afGe[542, 0] := 7.10000E+03; afGe[542, 1] := 1.09471E+00;
afGe[543, 0] := 7.15000E+03; afGe[543, 1] := 1.08126E+00;
afGe[544, 0] := 7.20000E+03; afGe[544, 1] := 1.06804E+00;
afGe[545, 0] := 7.25000E+03; afGe[545, 1] := 1.05510E+00;
afGe[546, 0] := 7.30000E+03; afGe[546, 1] := 1.04242E+00;
afGe[547, 0] := 7.35000E+03; afGe[547, 1] := 1.02997E+00;
afGe[548, 0] := 7.40000E+03; afGe[548, 1] := 1.01779E+00;
afGe[549, 0] := 7.45000E+03; afGe[549, 1] := 1.00585E+00;
afGe[550, 0] := 7.50000E+03; afGe[550, 1] := 9.94131E-01;
afGe[551, 0] := 7.55000E+03; afGe[551, 1] := 9.82627E-01;
afGe[552, 0] := 7.60000E+03; afGe[552, 1] := 9.71336E-01;
afGe[553, 0] := 7.65000E+03; afGe[553, 1] := 9.60268E-01;
afGe[554, 0] := 7.70000E+03; afGe[554, 1] := 9.49401E-01;
afGe[555, 0] := 7.75000E+03; afGe[555, 1] := 9.38730E-01;
afGe[556, 0] := 7.80000E+03; afGe[556, 1] := 9.28257E-01;
afGe[557, 0] := 7.85000E+03; afGe[557, 1] := 9.17976E-01;
afGe[558, 0] := 7.90000E+03; afGe[558, 1] := 9.07884E-01;
afGe[559, 0] := 7.95000E+03; afGe[559, 1] := 8.97970E-01;
afGe[560, 0] := 8.00000E+03; afGe[560, 1] := 8.88230E-01;
afGe[561, 0] := 8.05000E+03; afGe[561, 1] := 8.78666E-01;
afGe[562, 0] := 8.10000E+03; afGe[562, 1] := 8.69271E-01;
afGe[563, 0] := 8.15000E+03; afGe[563, 1] := 8.60037E-01;
afGe[564, 0] := 8.20000E+03; afGe[564, 1] := 8.50965E-01;
afGe[565, 0] := 8.25000E+03; afGe[565, 1] := 8.42050E-01;
afGe[566, 0] := 8.30000E+03; afGe[566, 1] := 8.33291E-01;
afGe[567, 0] := 8.35000E+03; afGe[567, 1] := 8.24682E-01;
afGe[568, 0] := 8.40000E+03; afGe[568, 1] := 8.16215E-01;
afGe[569, 0] := 8.45000E+03; afGe[569, 1] := 8.07894E-01;
afGe[570, 0] := 8.50000E+03; afGe[570, 1] := 7.99709E-01;
afGe[571, 0] := 8.55000E+03; afGe[571, 1] := 7.91659E-01;
afGe[572, 0] := 8.60000E+03; afGe[572, 1] := 7.83744E-01;
afGe[573, 0] := 8.65000E+03; afGe[573, 1] := 7.75957E-01;
afGe[574, 0] := 8.70000E+03; afGe[574, 1] := 7.68302E-01;
afGe[575, 0] := 8.75000E+03; afGe[575, 1] := 7.60770E-01;
afGe[576, 0] := 8.80000E+03; afGe[576, 1] := 7.53360E-01;
afGe[577, 0] := 8.85000E+03; afGe[577, 1] := 7.46013E-01;
afGe[578, 0] := 8.90000E+03; afGe[578, 1] := 7.38749E-01;
afGe[579, 0] := 8.95000E+03; afGe[579, 1] := 7.30771E-01;
afGe[580, 0] := 9.00000E+03; afGe[580, 1] := 7.22789E-01;
afGe[581, 0] := 9.05000E+03; afGe[581, 1] := 7.14945E-01;
afGe[582, 0] := 9.10000E+03; afGe[582, 1] := 7.07231E-01;
afGe[583, 0] := 9.15000E+03; afGe[583, 1] := 6.99649E-01;
afGe[584, 0] := 9.20000E+03; afGe[584, 1] := 6.92328E-01;
afGe[585, 0] := 9.25000E+03; afGe[585, 1] := 6.85282E-01;
afGe[586, 0] := 9.30000E+03; afGe[586, 1] := 6.78188E-01;
afGe[587, 0] := 9.35000E+03; afGe[587, 1] := 6.71112E-01;
afGe[588, 0] := 9.40000E+03; afGe[588, 1] := 6.64149E-01;
afGe[589, 0] := 9.45000E+03; afGe[589, 1] := 6.57295E-01;
afGe[590, 0] := 9.50000E+03; afGe[590, 1] := 6.50563E-01;
afGe[591, 0] := 9.55000E+03; afGe[591, 1] := 6.43937E-01;
afGe[592, 0] := 9.60000E+03; afGe[592, 1] := 6.37416E-01;
afGe[593, 0] := 9.65000E+03; afGe[593, 1] := 6.30996E-01;
afGe[594, 0] := 9.70000E+03; afGe[594, 1] := 6.24688E-01;
afGe[595, 0] := 9.75000E+03; afGe[595, 1] := 6.18478E-01;
afGe[596, 0] := 9.80000E+03; afGe[596, 1] := 6.12368E-01;
afGe[597, 0] := 9.85000E+03; afGe[597, 1] := 6.06352E-01;
afGe[598, 0] := 9.90000E+03; afGe[598, 1] := 6.00434E-01;
afGe[599, 0] := 9.95000E+03; afGe[599, 1] := 5.94607E-01;
afGe[600, 0] := 1.00000E+04; afGe[600, 1] := 5.88876E-01;
afGe[601, 0] := 1.00500E+04; afGe[601, 1] := 5.83234E-01;
afGe[602, 0] := 1.01000E+04; afGe[602, 1] := 5.77685E-01;
afGe[603, 0] := 1.01500E+04; afGe[603, 1] := 5.72222E-01;
afGe[604, 0] := 1.02000E+04; afGe[604, 1] := 5.66851E-01;
afGe[605, 0] := 1.02500E+04; afGe[605, 1] := 5.61562E-01;
afGe[606, 0] := 1.03000E+04; afGe[606, 1] := 5.56369E-01;
afGe[607, 0] := 1.03500E+04; afGe[607, 1] := 5.51255E-01;
afGe[608, 0] := 1.04000E+04; afGe[608, 1] := 5.46236E-01;
afGe[609, 0] := 1.04500E+04; afGe[609, 1] := 5.41292E-01;
afGe[610, 0] := 1.05000E+04; afGe[610, 1] := 5.36457E-01;
afGe[611, 0] := 1.05500E+04; afGe[611, 1] := 5.31690E-01;
afGe[612, 0] := 1.06000E+04; afGe[612, 1] := 5.27065E-01;
afGe[613, 0] := 1.06500E+04; afGe[613, 1] := 5.22501E-01;
afGe[614, 0] := 1.07000E+04; afGe[614, 1] := 5.18126E-01;
afGe[615, 0] := 1.07500E+04; afGe[615, 1] := 5.13819E-01;
afGe[616, 0] := 1.08000E+04; afGe[616, 1] := 5.09923E-01;
afGe[617, 0] := 1.08500E+04; afGe[617, 1] := 5.06168E-01;
afGe[618, 0] := 1.09000E+04; afGe[618, 1] := 5.03073E-01;
afGe[619, 0] := 1.09500E+04; afGe[619, 1] := 5.00360E-01;
afGe[620, 0] := 1.10000E+04; afGe[620, 1] := 5.00019E-01;
afGe[621, 0] := 1.10500E+04; afGe[621, 1] := 5.04812E-01;
afGe[622, 0] := 1.11000E+04; afGe[622, 1] := 8.05988E-01;
afGe[623, 0] := 1.11500E+04; afGe[623, 1] := 3.81021E+00;
afGe[624, 0] := 1.12000E+04; afGe[624, 1] := 3.78748E+00;
afGe[625, 0] := 1.12500E+04; afGe[625, 1] := 3.75455E+00;
afGe[626, 0] := 1.13000E+04; afGe[626, 1] := 3.72205E+00;
afGe[627, 0] := 1.13500E+04; afGe[627, 1] := 3.68862E+00;
afGe[628, 0] := 1.14000E+04; afGe[628, 1] := 3.65532E+00;
afGe[629, 0] := 1.14500E+04; afGe[629, 1] := 3.62229E+00;
afGe[630, 0] := 1.15000E+04; afGe[630, 1] := 3.58955E+00;
afGe[631, 0] := 1.15500E+04; afGe[631, 1] := 3.55724E+00;
afGe[632, 0] := 1.16000E+04; afGe[632, 1] := 3.52530E+00;
afGe[633, 0] := 1.16500E+04; afGe[633, 1] := 3.49379E+00;
afGe[634, 0] := 1.17000E+04; afGe[634, 1] := 3.46656E+00;
afGe[635, 0] := 1.17500E+04; afGe[635, 1] := 3.43984E+00;
afGe[636, 0] := 1.18000E+04; afGe[636, 1] := 3.41375E+00;
afGe[637, 0] := 1.18500E+04; afGe[637, 1] := 3.38816E+00;
afGe[638, 0] := 1.19000E+04; afGe[638, 1] := 3.36298E+00;
afGe[639, 0] := 1.19500E+04; afGe[639, 1] := 3.33838E+00;
afGe[640, 0] := 1.20000E+04; afGe[640, 1] := 3.31406E+00;
afGe[641, 0] := 1.20500E+04; afGe[641, 1] := 3.29036E+00;
afGe[642, 0] := 1.21000E+04; afGe[642, 1] := 3.26696E+00;
afGe[643, 0] := 1.21500E+04; afGe[643, 1] := 3.24400E+00;
afGe[644, 0] := 1.22000E+04; afGe[644, 1] := 3.22148E+00;
afGe[645, 0] := 1.22500E+04; afGe[645, 1] := 3.19922E+00;
afGe[646, 0] := 1.23000E+04; afGe[646, 1] := 3.17751E+00;
afGe[647, 0] := 1.23500E+04; afGe[647, 1] := 3.15603E+00;
afGe[648, 0] := 1.24000E+04; afGe[648, 1] := 3.13497E+00;
afGe[649, 0] := 1.24500E+04; afGe[649, 1] := 3.11425E+00;
afGe[650, 0] := 1.25000E+04; afGe[650, 1] := 3.09378E+00;
afGe[651, 0] := 1.25500E+04; afGe[651, 1] := 3.07372E+00;
afGe[652, 0] := 1.26000E+04; afGe[652, 1] := 3.05387E+00;
afGe[653, 0] := 1.26500E+04; afGe[653, 1] := 3.03436E+00;
afGe[654, 0] := 1.27000E+04; afGe[654, 1] := 3.01512E+00;
afGe[655, 0] := 1.27500E+04; afGe[655, 1] := 2.99610E+00;
afGe[656, 0] := 1.28000E+04; afGe[656, 1] := 2.97746E+00;
afGe[657, 0] := 1.28500E+04; afGe[657, 1] := 2.95901E+00;
afGe[658, 0] := 1.29000E+04; afGe[658, 1] := 2.94093E+00;
afGe[659, 0] := 1.29500E+04; afGe[659, 1] := 2.92318E+00;
afGe[660, 0] := 1.30000E+04; afGe[660, 1] := 2.90561E+00;
afGe[661, 0] := 1.30500E+04; afGe[661, 1] := 2.88816E+00;
afGe[662, 0] := 1.31000E+04; afGe[662, 1] := 2.87089E+00;
afGe[663, 0] := 1.31500E+04; afGe[663, 1] := 2.85383E+00;
afGe[664, 0] := 1.32000E+04; afGe[664, 1] := 2.83701E+00;
afGe[665, 0] := 1.32500E+04; afGe[665, 1] := 2.82035E+00;
afGe[666, 0] := 1.33000E+04; afGe[666, 1] := 2.80391E+00;
afGe[667, 0] := 1.33500E+04; afGe[667, 1] := 2.78766E+00;
afGe[668, 0] := 1.34000E+04; afGe[668, 1] := 2.77156E+00;
afGe[669, 0] := 1.34500E+04; afGe[669, 1] := 2.75570E+00;
afGe[670, 0] := 1.35000E+04; afGe[670, 1] := 2.73999E+00;
afGe[671, 0] := 1.35500E+04; afGe[671, 1] := 2.72446E+00;
afGe[672, 0] := 1.36000E+04; afGe[672, 1] := 2.70910E+00;
afGe[673, 0] := 1.36500E+04; afGe[673, 1] := 2.69388E+00;
afGe[674, 0] := 1.37000E+04; afGe[674, 1] := 2.67885E+00;
afGe[675, 0] := 1.37500E+04; afGe[675, 1] := 2.66397E+00;
afGe[676, 0] := 1.38000E+04; afGe[676, 1] := 2.64924E+00;
afGe[677, 0] := 1.38500E+04; afGe[677, 1] := 2.63463E+00;
afGe[678, 0] := 1.39000E+04; afGe[678, 1] := 2.62015E+00;
afGe[679, 0] := 1.39500E+04; afGe[679, 1] := 2.60582E+00;
afGe[680, 0] := 1.40000E+04; afGe[680, 1] := 2.59168E+00;
afGe[681, 0] := 1.40500E+04; afGe[681, 1] := 2.57766E+00;
afGe[682, 0] := 1.41000E+04; afGe[682, 1] := 2.56375E+00;
afGe[683, 0] := 1.41500E+04; afGe[683, 1] := 2.54995E+00;
afGe[684, 0] := 1.42000E+04; afGe[684, 1] := 2.53627E+00;
afGe[685, 0] := 1.42500E+04; afGe[685, 1] := 2.52274E+00;
afGe[686, 0] := 1.43000E+04; afGe[686, 1] := 2.50935E+00;
afGe[687, 0] := 1.43500E+04; afGe[687, 1] := 2.49607E+00;
afGe[688, 0] := 1.44000E+04; afGe[688, 1] := 2.48246E+00;
afGe[689, 0] := 1.44500E+04; afGe[689, 1] := 2.46887E+00;
afGe[690, 0] := 1.45000E+04; afGe[690, 1] := 2.45539E+00;
afGe[691, 0] := 1.45500E+04; afGe[691, 1] := 2.44152E+00;
afGe[692, 0] := 1.46000E+04; afGe[692, 1] := 2.42773E+00;
afGe[693, 0] := 1.46500E+04; afGe[693, 1] := 2.41406E+00;
afGe[694, 0] := 1.47000E+04; afGe[694, 1] := 2.40050E+00;
afGe[695, 0] := 1.47500E+04; afGe[695, 1] := 2.38705E+00;
afGe[696, 0] := 1.48000E+04; afGe[696, 1] := 2.37373E+00;
afGe[697, 0] := 1.48500E+04; afGe[697, 1] := 2.36048E+00;
afGe[698, 0] := 1.49000E+04; afGe[698, 1] := 2.34735E+00;
afGe[699, 0] := 1.49500E+04; afGe[699, 1] := 2.33433E+00;
afGe[700, 0] := 1.50000E+04; afGe[700, 1] := 2.32142E+00;
afGe[701, 0] := 1.50500E+04; afGe[701, 1] := 2.30862E+00;
afGe[702, 0] := 1.51000E+04; afGe[702, 1] := 2.29593E+00;
afGe[703, 0] := 1.51500E+04; afGe[703, 1] := 2.28331E+00;
afGe[704, 0] := 1.52000E+04; afGe[704, 1] := 2.27080E+00;
afGe[705, 0] := 1.52500E+04; afGe[705, 1] := 2.25840E+00;
afGe[706, 0] := 1.53000E+04; afGe[706, 1] := 2.24607E+00;
afGe[707, 0] := 1.53500E+04; afGe[707, 1] := 2.23385E+00;
afGe[708, 0] := 1.54000E+04; afGe[708, 1] := 2.22173E+00;
afGe[709, 0] := 1.54500E+04; afGe[709, 1] := 2.20971E+00;
afGe[710, 0] := 1.55000E+04; afGe[710, 1] := 2.19780E+00;
afGe[711, 0] := 1.55500E+04; afGe[711, 1] := 2.18598E+00;
afGe[712, 0] := 1.56000E+04; afGe[712, 1] := 2.17424E+00;
afGe[713, 0] := 1.56500E+04; afGe[713, 1] := 2.16259E+00;
afGe[714, 0] := 1.57000E+04; afGe[714, 1] := 2.15105E+00;
afGe[715, 0] := 1.57500E+04; afGe[715, 1] := 2.13954E+00;
afGe[716, 0] := 1.58000E+04; afGe[716, 1] := 2.12813E+00;
afGe[717, 0] := 1.58500E+04; afGe[717, 1] := 2.11681E+00;
afGe[718, 0] := 1.59000E+04; afGe[718, 1] := 2.10559E+00;
afGe[719, 0] := 1.59500E+04; afGe[719, 1] := 2.09446E+00;
afGe[720, 0] := 1.60000E+04; afGe[720, 1] := 2.08343E+00;
afGe[721, 0] := 1.60500E+04; afGe[721, 1] := 2.07247E+00;
afGe[722, 0] := 1.61000E+04; afGe[722, 1] := 2.06160E+00;
afGe[723, 0] := 1.61500E+04; afGe[723, 1] := 2.05081E+00;
afGe[724, 0] := 1.62000E+04; afGe[724, 1] := 2.04011E+00;
afGe[725, 0] := 1.62500E+04; afGe[725, 1] := 2.02947E+00;
afGe[726, 0] := 1.63000E+04; afGe[726, 1] := 2.01893E+00;
afGe[727, 0] := 1.63500E+04; afGe[727, 1] := 2.00847E+00;
afGe[728, 0] := 1.64000E+04; afGe[728, 1] := 1.99807E+00;
afGe[729, 0] := 1.64500E+04; afGe[729, 1] := 1.98776E+00;
afGe[730, 0] := 1.65000E+04; afGe[730, 1] := 1.97754E+00;
afGe[731, 0] := 1.65500E+04; afGe[731, 1] := 1.96738E+00;
afGe[732, 0] := 1.66000E+04; afGe[732, 1] := 1.95730E+00;
afGe[733, 0] := 1.66500E+04; afGe[733, 1] := 1.94730E+00;
afGe[734, 0] := 1.67000E+04; afGe[734, 1] := 1.93736E+00;
afGe[735, 0] := 1.67500E+04; afGe[735, 1] := 1.92747E+00;
afGe[736, 0] := 1.68000E+04; afGe[736, 1] := 1.91767E+00;
afGe[737, 0] := 1.68500E+04; afGe[737, 1] := 1.90794E+00;
afGe[738, 0] := 1.69000E+04; afGe[738, 1] := 1.89831E+00;
afGe[739, 0] := 1.69500E+04; afGe[739, 1] := 1.88875E+00;
afGe[740, 0] := 1.70000E+04; afGe[740, 1] := 1.87927E+00;
afGe[741, 0] := 1.70500E+04; afGe[741, 1] := 1.86983E+00;
afGe[742, 0] := 1.71000E+04; afGe[742, 1] := 1.86045E+00;
afGe[743, 0] := 1.71500E+04; afGe[743, 1] := 1.85115E+00;
afGe[744, 0] := 1.72000E+04; afGe[744, 1] := 1.84192E+00;
afGe[745, 0] := 1.72500E+04; afGe[745, 1] := 1.83276E+00;
afGe[746, 0] := 1.73000E+04; afGe[746, 1] := 1.82366E+00;
afGe[747, 0] := 1.73500E+04; afGe[747, 1] := 1.81464E+00;
afGe[748, 0] := 1.74000E+04; afGe[748, 1] := 1.80568E+00;
afGe[749, 0] := 1.74500E+04; afGe[749, 1] := 1.79679E+00;
afGe[750, 0] := 1.75000E+04; afGe[750, 1] := 1.78797E+00;
afGe[751, 0] := 1.75500E+04; afGe[751, 1] := 1.77921E+00;
afGe[752, 0] := 1.76000E+04; afGe[752, 1] := 1.77052E+00;
afGe[753, 0] := 1.76500E+04; afGe[753, 1] := 1.76189E+00;
afGe[754, 0] := 1.77000E+04; afGe[754, 1] := 1.75334E+00;
afGe[755, 0] := 1.77500E+04; afGe[755, 1] := 1.74484E+00;
afGe[756, 0] := 1.78000E+04; afGe[756, 1] := 1.73640E+00;
afGe[757, 0] := 1.78500E+04; afGe[757, 1] := 1.72804E+00;
afGe[758, 0] := 1.79000E+04; afGe[758, 1] := 1.71971E+00;
afGe[759, 0] := 1.79500E+04; afGe[759, 1] := 1.71144E+00;
afGe[760, 0] := 1.80000E+04; afGe[760, 1] := 1.70323E+00;
afGe[761, 0] := 1.80500E+04; afGe[761, 1] := 1.69509E+00;
afGe[762, 0] := 1.81000E+04; afGe[762, 1] := 1.68700E+00;
afGe[763, 0] := 1.81500E+04; afGe[763, 1] := 1.67897E+00;
afGe[764, 0] := 1.82000E+04; afGe[764, 1] := 1.67101E+00;
afGe[765, 0] := 1.82500E+04; afGe[765, 1] := 1.66309E+00;
afGe[766, 0] := 1.83000E+04; afGe[766, 1] := 1.65522E+00;
afGe[767, 0] := 1.83500E+04; afGe[767, 1] := 1.64740E+00;
afGe[768, 0] := 1.84000E+04; afGe[768, 1] := 1.63965E+00;
afGe[769, 0] := 1.84500E+04; afGe[769, 1] := 1.63195E+00;
afGe[770, 0] := 1.85000E+04; afGe[770, 1] := 1.62431E+00;
afGe[771, 0] := 1.85500E+04; afGe[771, 1] := 1.61673E+00;
afGe[772, 0] := 1.86000E+04; afGe[772, 1] := 1.60920E+00;
afGe[773, 0] := 1.86500E+04; afGe[773, 1] := 1.60174E+00;
afGe[774, 0] := 1.87000E+04; afGe[774, 1] := 1.59432E+00;
afGe[775, 0] := 1.87500E+04; afGe[775, 1] := 1.58697E+00;
afGe[776, 0] := 1.88000E+04; afGe[776, 1] := 1.57966E+00;
afGe[777, 0] := 1.88500E+04; afGe[777, 1] := 1.57239E+00;
afGe[778, 0] := 1.89000E+04; afGe[778, 1] := 1.56517E+00;
afGe[779, 0] := 1.89500E+04; afGe[779, 1] := 1.55800E+00;
afGe[780, 0] := 1.90000E+04; afGe[780, 1] := 1.55089E+00;
afGe[781, 0] := 1.90500E+04; afGe[781, 1] := 1.54384E+00;
afGe[782, 0] := 1.91000E+04; afGe[782, 1] := 1.53684E+00;
afGe[783, 0] := 1.91500E+04; afGe[783, 1] := 1.52988E+00;
afGe[784, 0] := 1.92000E+04; afGe[784, 1] := 1.52297E+00;
afGe[785, 0] := 1.92500E+04; afGe[785, 1] := 1.51610E+00;
afGe[786, 0] := 1.93000E+04; afGe[786, 1] := 1.50928E+00;
afGe[787, 0] := 1.93500E+04; afGe[787, 1] := 1.50251E+00;
afGe[788, 0] := 1.94000E+04; afGe[788, 1] := 1.49580E+00;
afGe[789, 0] := 1.94500E+04; afGe[789, 1] := 1.48913E+00;
afGe[790, 0] := 1.95000E+04; afGe[790, 1] := 1.48251E+00;
afGe[791, 0] := 1.95500E+04; afGe[791, 1] := 1.47594E+00;
afGe[792, 0] := 1.96000E+04; afGe[792, 1] := 1.46941E+00;
afGe[793, 0] := 1.96500E+04; afGe[793, 1] := 1.46292E+00;
afGe[794, 0] := 1.97000E+04; afGe[794, 1] := 1.45647E+00;
afGe[795, 0] := 1.97500E+04; afGe[795, 1] := 1.45007E+00;
afGe[796, 0] := 1.98000E+04; afGe[796, 1] := 1.44371E+00;
afGe[797, 0] := 1.98500E+04; afGe[797, 1] := 1.43738E+00;
afGe[798, 0] := 1.99000E+04; afGe[798, 1] := 1.43111E+00;
afGe[799, 0] := 1.99500E+04; afGe[799, 1] := 1.42487E+00;
afGe[800, 0] := 2.00000E+04; afGe[800, 1] := 1.41870E+00;
afGe[801, 0] := 2.00500E+04; afGe[801, 1] := 1.41257E+00;
afGe[802, 0] := 2.01000E+04; afGe[802, 1] := 1.40648E+00;
afGe[803, 0] := 2.01500E+04; afGe[803, 1] := 1.40043E+00;
afGe[804, 0] := 2.02000E+04; afGe[804, 1] := 1.39442E+00;
afGe[805, 0] := 2.02500E+04; afGe[805, 1] := 1.38845E+00;
afGe[806, 0] := 2.03000E+04; afGe[806, 1] := 1.38252E+00;
afGe[807, 0] := 2.03500E+04; afGe[807, 1] := 1.37663E+00;
afGe[808, 0] := 2.04000E+04; afGe[808, 1] := 1.37077E+00;
afGe[809, 0] := 2.04500E+04; afGe[809, 1] := 1.36496E+00;
afGe[810, 0] := 2.05000E+04; afGe[810, 1] := 1.35918E+00;
afGe[811, 0] := 2.05500E+04; afGe[811, 1] := 1.35344E+00;
afGe[812, 0] := 2.06000E+04; afGe[812, 1] := 1.34774E+00;
afGe[813, 0] := 2.06500E+04; afGe[813, 1] := 1.34208E+00;
afGe[814, 0] := 2.07000E+04; afGe[814, 1] := 1.33645E+00;
afGe[815, 0] := 2.07500E+04; afGe[815, 1] := 1.33086E+00;
afGe[816, 0] := 2.08000E+04; afGe[816, 1] := 1.32531E+00;
afGe[817, 0] := 2.08500E+04; afGe[817, 1] := 1.31979E+00;
afGe[818, 0] := 2.09000E+04; afGe[818, 1] := 1.31431E+00;
afGe[819, 0] := 2.09500E+04; afGe[819, 1] := 1.30887E+00;
afGe[820, 0] := 2.10000E+04; afGe[820, 1] := 1.30347E+00;
afGe[821, 0] := 2.10500E+04; afGe[821, 1] := 1.29809E+00;
afGe[822, 0] := 2.11000E+04; afGe[822, 1] := 1.29276E+00;
afGe[823, 0] := 2.11500E+04; afGe[823, 1] := 1.28746E+00;
afGe[824, 0] := 2.12000E+04; afGe[824, 1] := 1.28219E+00;
afGe[825, 0] := 2.12500E+04; afGe[825, 1] := 1.27696E+00;
afGe[826, 0] := 2.13000E+04; afGe[826, 1] := 1.27177E+00;
afGe[827, 0] := 2.13500E+04; afGe[827, 1] := 1.26661E+00;
afGe[828, 0] := 2.14000E+04; afGe[828, 1] := 1.26148E+00;
afGe[829, 0] := 2.14500E+04; afGe[829, 1] := 1.25639E+00;
afGe[830, 0] := 2.15000E+04; afGe[830, 1] := 1.25133E+00;
afGe[831, 0] := 2.15500E+04; afGe[831, 1] := 1.24630E+00;
afGe[832, 0] := 2.16000E+04; afGe[832, 1] := 1.24130E+00;
afGe[833, 0] := 2.16500E+04; afGe[833, 1] := 1.23632E+00;
afGe[834, 0] := 2.17000E+04; afGe[834, 1] := 1.23138E+00;
afGe[835, 0] := 2.17500E+04; afGe[835, 1] := 1.22646E+00;
afGe[836, 0] := 2.18000E+04; afGe[836, 1] := 1.22157E+00;
afGe[837, 0] := 2.18500E+04; afGe[837, 1] := 1.21674E+00;
afGe[838, 0] := 2.19000E+04; afGe[838, 1] := 1.21195E+00;
afGe[839, 0] := 2.19500E+04; afGe[839, 1] := 1.20718E+00;
afGe[840, 0] := 2.20000E+04; afGe[840, 1] := 1.20245E+00;
afGe[841, 0] := 2.20500E+04; afGe[841, 1] := 1.19772E+00;
afGe[842, 0] := 2.21000E+04; afGe[842, 1] := 1.19301E+00;
afGe[843, 0] := 2.21500E+04; afGe[843, 1] := 1.18833E+00;
afGe[844, 0] := 2.22000E+04; afGe[844, 1] := 1.18367E+00;
afGe[845, 0] := 2.22500E+04; afGe[845, 1] := 1.17904E+00;
afGe[846, 0] := 2.23000E+04; afGe[846, 1] := 1.17432E+00;
afGe[847, 0] := 2.23500E+04; afGe[847, 1] := 1.16963E+00;
afGe[848, 0] := 2.24000E+04; afGe[848, 1] := 1.16496E+00;
afGe[849, 0] := 2.24500E+04; afGe[849, 1] := 1.16032E+00;
afGe[850, 0] := 2.25000E+04; afGe[850, 1] := 1.15572E+00;
afGe[851, 0] := 2.25500E+04; afGe[851, 1] := 1.15115E+00;
afGe[852, 0] := 2.26000E+04; afGe[852, 1] := 1.14661E+00;
afGe[853, 0] := 2.26500E+04; afGe[853, 1] := 1.14209E+00;
afGe[854, 0] := 2.27000E+04; afGe[854, 1] := 1.13760E+00;
afGe[855, 0] := 2.27500E+04; afGe[855, 1] := 1.13313E+00;
afGe[856, 0] := 2.28000E+04; afGe[856, 1] := 1.12868E+00;
afGe[857, 0] := 2.28500E+04; afGe[857, 1] := 1.12426E+00;
afGe[858, 0] := 2.29000E+04; afGe[858, 1] := 1.11987E+00;
afGe[859, 0] := 2.29500E+04; afGe[859, 1] := 1.11552E+00;
afGe[860, 0] := 2.30000E+04; afGe[860, 1] := 1.11121E+00;
afGe[861, 0] := 2.30500E+04; afGe[861, 1] := 1.10693E+00;
afGe[862, 0] := 2.31000E+04; afGe[862, 1] := 1.10268E+00;
afGe[863, 0] := 2.31500E+04; afGe[863, 1] := 1.09845E+00;
afGe[864, 0] := 2.32000E+04; afGe[864, 1] := 1.09421E+00;
afGe[865, 0] := 2.32500E+04; afGe[865, 1] := 1.09000E+00;
afGe[866, 0] := 2.33000E+04; afGe[866, 1] := 1.08581E+00;
afGe[867, 0] := 2.33500E+04; afGe[867, 1] := 1.08165E+00;
afGe[868, 0] := 2.34000E+04; afGe[868, 1] := 1.07752E+00;
afGe[869, 0] := 2.34500E+04; afGe[869, 1] := 1.07342E+00;
afGe[870, 0] := 2.35000E+04; afGe[870, 1] := 1.06935E+00;
afGe[871, 0] := 2.35500E+04; afGe[871, 1] := 1.06530E+00;
afGe[872, 0] := 2.36000E+04; afGe[872, 1] := 1.06127E+00;
afGe[873, 0] := 2.36500E+04; afGe[873, 1] := 1.05728E+00;
afGe[874, 0] := 2.37000E+04; afGe[874, 1] := 1.05331E+00;
afGe[875, 0] := 2.37500E+04; afGe[875, 1] := 1.04937E+00;
afGe[876, 0] := 2.38000E+04; afGe[876, 1] := 1.04545E+00;
afGe[877, 0] := 2.38500E+04; afGe[877, 1] := 1.04155E+00;
afGe[878, 0] := 2.39000E+04; afGe[878, 1] := 1.03765E+00;
afGe[879, 0] := 2.39500E+04; afGe[879, 1] := 1.03377E+00;
afGe[880, 0] := 2.40000E+04; afGe[880, 1] := 1.02992E+00;
afGe[881, 0] := 2.40500E+04; afGe[881, 1] := 1.02609E+00;
afGe[882, 0] := 2.41000E+04; afGe[882, 1] := 1.02228E+00;
afGe[883, 0] := 2.41500E+04; afGe[883, 1] := 1.01850E+00;
afGe[884, 0] := 2.42000E+04; afGe[884, 1] := 1.01475E+00;
afGe[885, 0] := 2.42500E+04; afGe[885, 1] := 1.01102E+00;
afGe[886, 0] := 2.43000E+04; afGe[886, 1] := 1.00731E+00;
afGe[887, 0] := 2.43500E+04; afGe[887, 1] := 1.00363E+00;
afGe[888, 0] := 2.44000E+04; afGe[888, 1] := 9.99963E-01;
afGe[889, 0] := 2.44500E+04; afGe[889, 1] := 9.96321E-01;
afGe[890, 0] := 2.45000E+04; afGe[890, 1] := 9.92698E-01;
afGe[891, 0] := 2.45500E+04; afGe[891, 1] := 9.89097E-01;
afGe[892, 0] := 2.46000E+04; afGe[892, 1] := 9.85513E-01;
afGe[893, 0] := 2.46500E+04; afGe[893, 1] := 9.81948E-01;
afGe[894, 0] := 2.47000E+04; afGe[894, 1] := 9.78402E-01;
afGe[895, 0] := 2.47500E+04; afGe[895, 1] := 9.74877E-01;
afGe[896, 0] := 2.48000E+04; afGe[896, 1] := 9.71371E-01;
afGe[897, 0] := 2.48500E+04; afGe[897, 1] := 9.67886E-01;
afGe[898, 0] := 2.49000E+04; afGe[898, 1] := 9.64420E-01;
afGe[899, 0] := 2.49500E+04; afGe[899, 1] := 9.60973E-01;
afGe[900, 0] := 2.50000E+04; afGe[900, 1] := 9.57546E-01;
afGe[901, 0] := 2.50500E+04; afGe[901, 1] := 9.54138E-01;
afGe[902, 0] := 2.51000E+04; afGe[902, 1] := 9.50750E-01;
afGe[903, 0] := 2.51500E+04; afGe[903, 1] := 9.47381E-01;
afGe[904, 0] := 2.52000E+04; afGe[904, 1] := 9.44031E-01;
afGe[905, 0] := 2.52500E+04; afGe[905, 1] := 9.40700E-01;
afGe[906, 0] := 2.53000E+04; afGe[906, 1] := 9.37386E-01;
afGe[907, 0] := 2.53500E+04; afGe[907, 1] := 9.34091E-01;
afGe[908, 0] := 2.54000E+04; afGe[908, 1] := 9.30813E-01;
afGe[909, 0] := 2.54500E+04; afGe[909, 1] := 9.27553E-01;
afGe[910, 0] := 2.55000E+04; afGe[910, 1] := 9.24310E-01;
afGe[911, 0] := 2.55500E+04; afGe[911, 1] := 9.21086E-01;
afGe[912, 0] := 2.56000E+04; afGe[912, 1] := 9.17879E-01;
afGe[913, 0] := 2.56500E+04; afGe[913, 1] := 9.14689E-01;
afGe[914, 0] := 2.57000E+04; afGe[914, 1] := 9.11516E-01;
afGe[915, 0] := 2.57500E+04; afGe[915, 1] := 9.08361E-01;
afGe[916, 0] := 2.58000E+04; afGe[916, 1] := 9.05223E-01;
afGe[917, 0] := 2.58500E+04; afGe[917, 1] := 9.02101E-01;
afGe[918, 0] := 2.59000E+04; afGe[918, 1] := 8.98995E-01;
afGe[919, 0] := 2.59500E+04; afGe[919, 1] := 8.95907E-01;
afGe[920, 0] := 2.60000E+04; afGe[920, 1] := 8.92834E-01;
afGe[921, 0] := 2.60500E+04; afGe[921, 1] := 8.89778E-01;
afGe[922, 0] := 2.61000E+04; afGe[922, 1] := 8.86738E-01;
afGe[923, 0] := 2.61500E+04; afGe[923, 1] := 8.83713E-01;
afGe[924, 0] := 2.62000E+04; afGe[924, 1] := 8.80703E-01;
afGe[925, 0] := 2.62500E+04; afGe[925, 1] := 8.77710E-01;
afGe[926, 0] := 2.63000E+04; afGe[926, 1] := 8.74732E-01;
afGe[927, 0] := 2.63500E+04; afGe[927, 1] := 8.71770E-01;
afGe[928, 0] := 2.64000E+04; afGe[928, 1] := 8.68825E-01;
afGe[929, 0] := 2.64500E+04; afGe[929, 1] := 8.65895E-01;
afGe[930, 0] := 2.65000E+04; afGe[930, 1] := 8.62981E-01;
afGe[931, 0] := 2.65500E+04; afGe[931, 1] := 8.60082E-01;
afGe[932, 0] := 2.66000E+04; afGe[932, 1] := 8.57198E-01;
afGe[933, 0] := 2.66500E+04; afGe[933, 1] := 8.54248E-01;
afGe[934, 0] := 2.67000E+04; afGe[934, 1] := 8.51287E-01;
afGe[935, 0] := 2.67500E+04; afGe[935, 1] := 8.48343E-01;
afGe[936, 0] := 2.68000E+04; afGe[936, 1] := 8.45413E-01;
afGe[937, 0] := 2.68500E+04; afGe[937, 1] := 8.42500E-01;
afGe[938, 0] := 2.69000E+04; afGe[938, 1] := 8.39582E-01;
afGe[939, 0] := 2.69500E+04; afGe[939, 1] := 8.36652E-01;
afGe[940, 0] := 2.70000E+04; afGe[940, 1] := 8.33739E-01;
afGe[941, 0] := 2.70500E+04; afGe[941, 1] := 8.30841E-01;
afGe[942, 0] := 2.71000E+04; afGe[942, 1] := 8.27958E-01;
afGe[943, 0] := 2.71500E+04; afGe[943, 1] := 8.25091E-01;
afGe[944, 0] := 2.72000E+04; afGe[944, 1] := 8.22237E-01;
afGe[945, 0] := 2.72500E+04; afGe[945, 1] := 8.19398E-01;
afGe[946, 0] := 2.73000E+04; afGe[946, 1] := 8.16574E-01;
afGe[947, 0] := 2.73500E+04; afGe[947, 1] := 8.13765E-01;
afGe[948, 0] := 2.74000E+04; afGe[948, 1] := 8.10971E-01;
afGe[949, 0] := 2.74500E+04; afGe[949, 1] := 8.08192E-01;
afGe[950, 0] := 2.75000E+04; afGe[950, 1] := 8.05428E-01;
afGe[951, 0] := 2.75500E+04; afGe[951, 1] := 8.02678E-01;
afGe[952, 0] := 2.76000E+04; afGe[952, 1] := 7.99943E-01;
afGe[953, 0] := 2.76500E+04; afGe[953, 1] := 7.97222E-01;
afGe[954, 0] := 2.77000E+04; afGe[954, 1] := 7.94515E-01;
afGe[955, 0] := 2.77500E+04; afGe[955, 1] := 7.91825E-01;
afGe[956, 0] := 2.78000E+04; afGe[956, 1] := 7.89148E-01;
afGe[957, 0] := 2.78500E+04; afGe[957, 1] := 7.86485E-01;
afGe[958, 0] := 2.79000E+04; afGe[958, 1] := 7.83836E-01;
afGe[959, 0] := 2.79500E+04; afGe[959, 1] := 7.81200E-01;
afGe[960, 0] := 2.80000E+04; afGe[960, 1] := 7.78577E-01;
afGe[961, 0] := 2.80500E+04; afGe[961, 1] := 7.75966E-01;
afGe[962, 0] := 2.81000E+04; afGe[962, 1] := 7.73368E-01;
afGe[963, 0] := 2.81500E+04; afGe[963, 1] := 7.70784E-01;
afGe[964, 0] := 2.82000E+04; afGe[964, 1] := 7.68213E-01;
afGe[965, 0] := 2.82500E+04; afGe[965, 1] := 7.65655E-01;
afGe[966, 0] := 2.83000E+04; afGe[966, 1] := 7.63112E-01;
afGe[967, 0] := 2.83500E+04; afGe[967, 1] := 7.60582E-01;
afGe[968, 0] := 2.84000E+04; afGe[968, 1] := 7.58064E-01;
afGe[969, 0] := 2.84500E+04; afGe[969, 1] := 7.55560E-01;
afGe[970, 0] := 2.85000E+04; afGe[970, 1] := 7.53068E-01;
afGe[971, 0] := 2.85500E+04; afGe[971, 1] := 7.50589E-01;
afGe[972, 0] := 2.86000E+04; afGe[972, 1] := 7.48121E-01;
afGe[973, 0] := 2.86500E+04; afGe[973, 1] := 7.45666E-01;
afGe[974, 0] := 2.87000E+04; afGe[974, 1] := 7.43223E-01;
afGe[975, 0] := 2.87500E+04; afGe[975, 1] := 7.40793E-01;
afGe[976, 0] := 2.88000E+04; afGe[976, 1] := 7.38375E-01;
afGe[977, 0] := 2.88500E+04; afGe[977, 1] := 7.35969E-01;
afGe[978, 0] := 2.89000E+04; afGe[978, 1] := 7.33575E-01;
afGe[979, 0] := 2.89500E+04; afGe[979, 1] := 7.31193E-01;
afGe[980, 0] := 2.90000E+04; afGe[980, 1] := 7.28822E-01;
afGe[981, 0] := 2.90500E+04; afGe[981, 1] := 7.26464E-01;
afGe[982, 0] := 2.91000E+04; afGe[982, 1] := 7.24117E-01;
afGe[983, 0] := 2.91500E+04; afGe[983, 1] := 7.21783E-01;
afGe[984, 0] := 2.92000E+04; afGe[984, 1] := 7.19460E-01;
afGe[985, 0] := 2.92500E+04; afGe[985, 1] := 7.17149E-01;
afGe[986, 0] := 2.93000E+04; afGe[986, 1] := 7.14849E-01;
afGe[987, 0] := 2.93500E+04; afGe[987, 1] := 7.12560E-01;
afGe[988, 0] := 2.94000E+04; afGe[988, 1] := 7.10283E-01;
afGe[989, 0] := 2.94500E+04; afGe[989, 1] := 7.08017E-01;
afGe[990, 0] := 2.95000E+04; afGe[990, 1] := 7.05762E-01;
afGe[991, 0] := 2.95500E+04; afGe[991, 1] := 7.03518E-01;
afGe[992, 0] := 2.96000E+04; afGe[992, 1] := 7.01285E-01;
afGe[993, 0] := 2.96500E+04; afGe[993, 1] := 6.99063E-01;
afGe[994, 0] := 2.97000E+04; afGe[994, 1] := 6.96851E-01;
afGe[995, 0] := 2.97500E+04; afGe[995, 1] := 6.94649E-01;
afGe[996, 0] := 2.98000E+04; afGe[996, 1] := 6.92459E-01;
afGe[997, 0] := 2.98500E+04; afGe[997, 1] := 6.90278E-01;
afGe[998, 0] := 2.99000E+04; afGe[998, 1] := 6.88108E-01;
afGe[999, 0] := 2.99500E+04; afGe[999, 1] := 6.85949E-01;

// Element = C

